# EPICS autosave request: soft_iocs/meas_comp/iocBoot/iocmeas_comp_ctr/ao.req
$(P)$(R).VAL
$(P)$(R).DRVH
$(P)$(R).DRVL
$(P)$(R).DESC
$(P)$(R).EGU
$(P)$(R).PREC
